(* IEC 61131-3 sources: PLC_MotorControl/src, 2 files *)

(* ---- configuration.st ---- *)
// Configuration settings for PLC Motor Control
VAR_GLOBAL
    // Add global variables here if necessary
END_VAR

(* ---- MotorControl.st ---- *)
// Motor Control Logic
FUNCTION_BLOCK MotorControl
VAR_INPUT
    StartButton: BOOL; // Input for start button
    StopButton: BOOL;  // Input for stop button
END_VAR

VAR_OUTPUT
    MotorRunning: BOOL; // Output to motor control
END_VAR

// Main program logic
IF StartButton AND NOT MotorRunning THEN
    MotorRunning := TRUE;
ELSIF StopButton THEN
    MotorRunning := FALSE;
END_IF;

END_FUNCTION_BLOCK
